Fanuc KAREL source: kt00586.KL

-- PROVISIONAL review KL for V940-1; original PC SHA256 a71c450265876c964a89675ace3e4a596b4b845aeb4b025aa15a98b5216c555f
-- Incomplete behavior may be omitted. Consult companion uncertainty JSON. Do not deploy.
PROGRAM KT00586
%NOLOCKGROUP
VAR
  I1 : INTEGER
-- UNRESOLVED_DECL V2 type=000013
-- UNRESOLVED_DECL OUT type=000013
BEGIN
  -- V9_ZERO_TABLE_METADATA_HINT layout=0001; no indexed target words; source/name/runtime held
  -- UNRESOLVED_PC offsets 5-16; opcodes 2E,23
  -- UNRESOLVED_PC offsets 21-36; opcodes 2E,22,32,35
  -- UNRESOLVED_PC offsets 41-63; opcodes 21,49,8F,4A
  -- UNRESOLVED_PC offsets 68-72; opcodes 7F
END KT00586
